GLOBALCONSTANTS DataPanel_MI_DO (* DataPanel Modules with medium IO density DO constants *)
  (* Standard: 61499-1; Description: Copyright (c) 2024 HR Agrartechnik GmbH This program and the accompanying materials are made available under the terms of the Eclipse Public License 2.0 which is available at https://www.eclipse.org/legal/epl-2.0/ SPDX-License-Identifier: EPL-2.0 *)
  (* Version 1.0, 2024-01-25, Franz Höpfinger, HR Agrartechnik GmbH *)
  PACKAGE DataPanel::io::MI::DQ;
  VAR_GLOBAL CONSTANT
    DigitalOutput_1A : DataPanel::io::MI::DQ::DataPanel_MI_DO_S := (Pin := 1);
    DigitalOutput_1B : DataPanel::io::MI::DQ::DataPanel_MI_DO_S := (Pin := 2);
    DigitalOutput_2A : DataPanel::io::MI::DQ::DataPanel_MI_DO_S := (Pin := 3);
    DigitalOutput_2B : DataPanel::io::MI::DQ::DataPanel_MI_DO_S := (Pin := 4);
    DigitalOutput_3A : DataPanel::io::MI::DQ::DataPanel_MI_DO_S := (Pin := 5);
    DigitalOutput_3B : DataPanel::io::MI::DQ::DataPanel_MI_DO_S := (Pin := 6);
    DigitalOutput_4A : DataPanel::io::MI::DQ::DataPanel_MI_DO_S := (Pin := 7);
    DigitalOutput_4B : DataPanel::io::MI::DQ::DataPanel_MI_DO_S := (Pin := 8);
    DigitalOutput_5A : DataPanel::io::MI::DQ::DataPanel_MI_DO_S := (Pin := 9);
    DigitalOutput_5B : DataPanel::io::MI::DQ::DataPanel_MI_DO_S := (Pin := 10);
    DigitalOutput_6A : DataPanel::io::MI::DQ::DataPanel_MI_DO_S := (Pin := 11);
    DigitalOutput_6B : DataPanel::io::MI::DQ::DataPanel_MI_DO_S := (Pin := 12);
    DigitalOutput_7A : DataPanel::io::MI::DQ::DataPanel_MI_DO_S := (Pin := 13);
    DigitalOutput_7B : DataPanel::io::MI::DQ::DataPanel_MI_DO_S := (Pin := 14);
    DigitalOutput_8A : DataPanel::io::MI::DQ::DataPanel_MI_DO_S := (Pin := 15);
    DigitalOutput_8B : DataPanel::io::MI::DQ::DataPanel_MI_DO_S := (Pin := 16);
    Input_Power_Port_5 : DataPanel::io::MI::DQ::DataPanel_MI_DO_S := (Pin := 17);
    Input_Power_Port_6 : DataPanel::io::MI::DQ::DataPanel_MI_DO_S := (Pin := 18);
    Input_Power_Port_7 : DataPanel::io::MI::DQ::DataPanel_MI_DO_S := (Pin := 19);
    Input_Power_Port_8 : DataPanel::io::MI::DQ::DataPanel_MI_DO_S := (Pin := 20);
    Invalid : DataPanel::io::MI::DQ::DataPanel_MI_DO_S := (Pin := 255);
  END_VAR
END_GLOBALCONSTANTS
